# EPICS substitutions: iocBoot/iocxxx/picMot.substitutions
file ipApp/Db/picos.db
{
pattern
{P,      pChan,       DESC,          serChan }
{xxx:, 	 111,         pMotor111,        1    }
{xxx:, 	 112,         pMotor112,        1    }
{xxx:, 	 113,         pMotor113,        1    }

{xxx:, 	 121,         pMotor121,        1    }
{xxx:, 	 122,         pMotor122,        1    }
{xxx:, 	 123,         pMotor123,        1    }

{xxx:, 	 131,         pMotor131,        1    }
{xxx:, 	 132,         pMotor132,        1    }
{xxx:, 	 133,         pMotor133,        1    }

{xxx:, 	 141,         pMotor141,        1    }
{xxx:, 	 142,         pMotor142,        1    }
{xxx:, 	 143,         pMotor143,        1    }

{xxx:, 	 211,         pMotor211,        1    }
{xxx:, 	 212,         pMotor212,        1    }
{xxx:, 	 213,         pMotor213,        1    }

{xxx:, 	 221,         pMotor221,        1    }
{xxx:, 	 222,         pMotor222,        1    }
{xxx:, 	 223,         pMotor223,        1    }

{xxx:, 	 231,         pMotor231,        1    }
{xxx:, 	 232,         pMotor232,        1    }
{xxx:, 	 233,         pMotor233,        1    }

{xxx:, 	 241,         pMotor241,        1    }
{xxx:, 	 242,         pMotor242,        1    }
{xxx:, 	 243,         pMotor243,        1    }

}
